(* Logix 5000 project; controller STAT 1756-L72 rev 20.12; software revision 20.04; part 21 of 34 *)
(* tags used below, declared in another part *)
   B10 : DINT[20];
   B14 : DINT[30];
   B17 : DINT[30];
   B3 : DINT[256];
   B9 : DINT[40];
   def1bassin : DINT;
   def2bassin : DINT;
   F8 : REAL[256];
   I10_000_Bit07 : ALIAS FOR I10[0].7;   // Hand Automaat CL8
   I19_000_Bit07 : ALIAS FOR I19[0].7;   // LACK DETECTIE H2SO4
   I1_001_Bit15 : ALIAS FOR I1[1].15;
   I1_008_Bit01 : ALIAS FOR I1[8].1;   // Hand Automaat stormbekken
   I1_016_Bit01 : ALIAS FOR I1[16].1;   // CL2 Hamd /Autom
   I1_017_Bit01 : ALIAS FOR I1[17].1;   // CL3 Hamd /Autom
   I1_018_Bit01 : ALIAS FOR I1[18].1;   // CL4 Hamd /Autom
   I2 : INT[2];
   I3 : INT[2];
   I4 : INT[2];
   I5 : INT[2];
   I6 : INT[2];
   I7 : INT[2];
   I8 : INT[2];
   I9_000_Bit09 : ALIAS FOR I9[0].9;   // Hand_Auto CL7
   N11 : DINT[150];
   N12 : DINT[230];
   N13 : DINT[230];
   N26 : DINT[256];
   N7 : DINT[255];
   O12 : INT[2];
   O13 : INT[2];
   O14 : INT[2];
   O15 : INT[2];
   O18 : INT[2];
   S : INT[164];
   T4 : TIMER[200];
(* ibt, continued *)

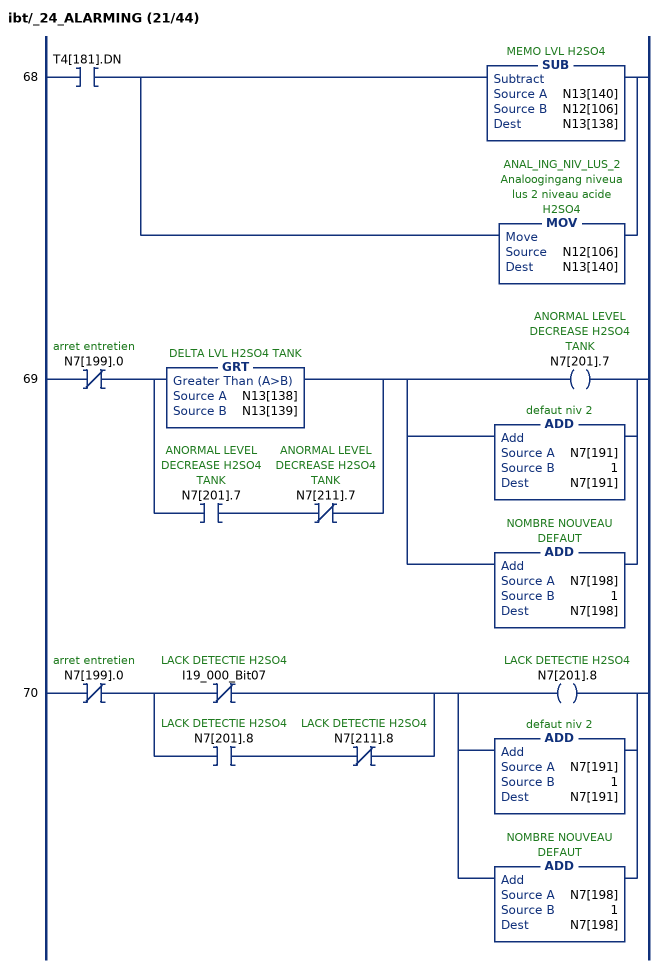
   [picture p391: ibt/_24_ALARMING rungs 68-70]
   68: XIC(T4[181].DN)[SUB(N13[140],N12[106],N13[138]) ,MOV(N12[106],N13[140]) ];
   69: XIO(N7[199].0)[GRT(N13[138],N13[139]) ,XIC(N7[201].7) XIO(N7[211].7) ][OTE(N7[201].7) ,ADD(N7[191],1,N7[191]) ,ADD(N7[198],1,N7[198]) ];
   70: XIO(N7[199].0)[XIO(I19_000_Bit07) ,XIC(N7[201].8) XIO(N7[211].8) ][OTE(N7[201].8) ,ADD(N7[191],1,N7[191]) ,ADD(N7[198],1,N7[198]) ];
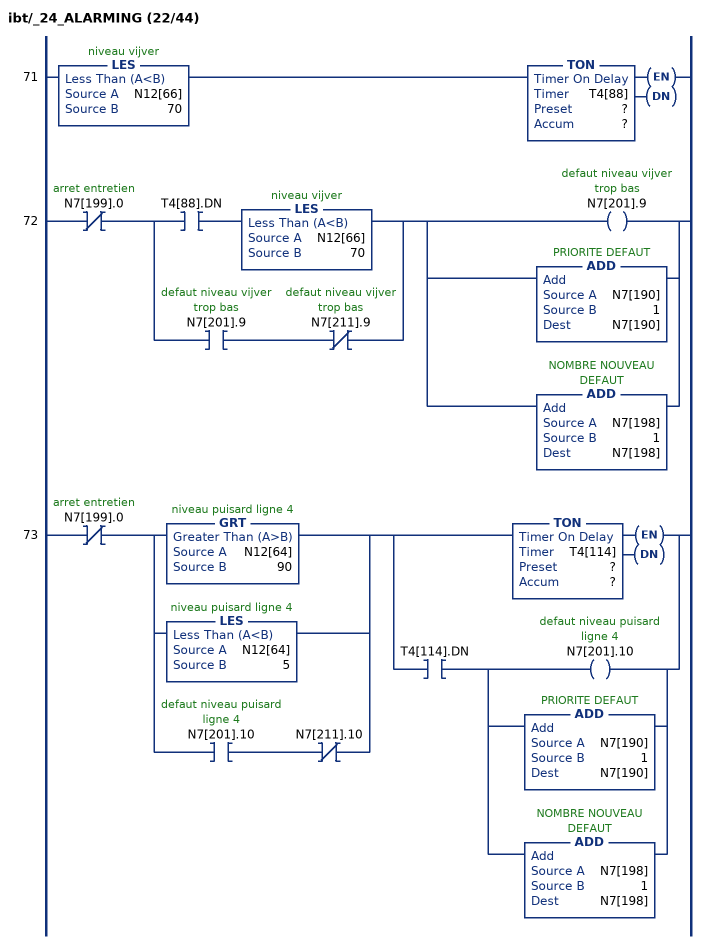
   71: LES(N12[66],70)TON(T4[88],?,?);
   72: XIO(N7[199].0)[XIC(T4[88].DN) LES(N12[66],70) ,XIC(N7[201].9) XIO(N7[211].9) ][OTE(N7[201].9) ,ADD(N7[190],1,N7[190]) ,ADD(N7[198],1,N7[198]) ];
   73: XIO(N7[199].0)[GRT(N12[64],90) ,LES(N12[64],5) ,XIC(N7[201].10) XIO(N7[211].10) ][TON(T4[114],?,?) ,XIC(T4[114].DN) [OTE(N7[201].10) ,ADD(N7[190],1,N7[190]) ,ADD(N7[198],1,N7[198]) ] ];
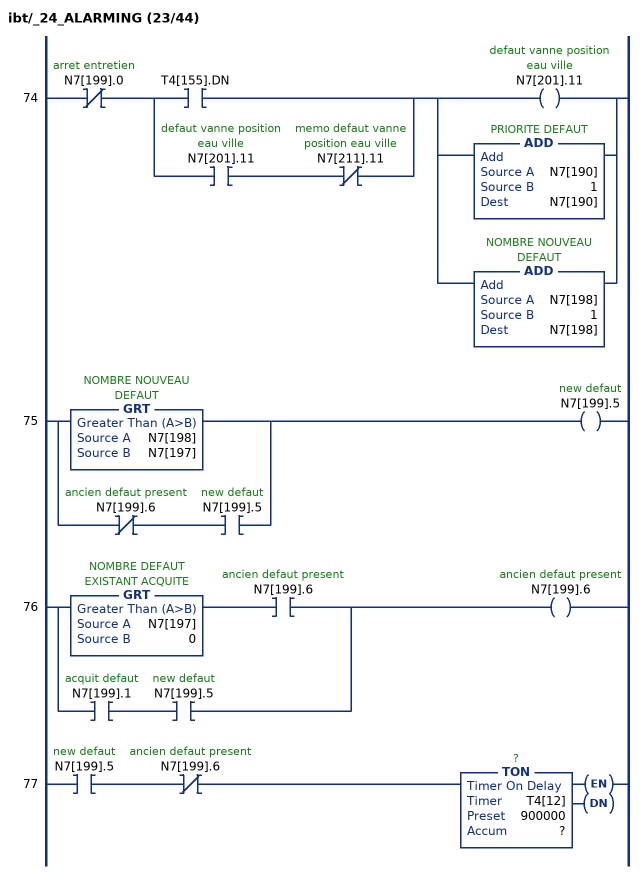
   74: XIO(N7[199].0)[XIC(T4[155].DN) ,XIC(N7[201].11) XIO(N7[211].11) ][OTE(N7[201].11) ,ADD(N7[190],1,N7[190]) ,ADD(N7[198],1,N7[198]) ];
   75: [GRT(N7[198],N7[197]) ,XIO(N7[199].6) XIC(N7[199].5) ]OTE(N7[199].5);
   76: [GRT(N7[197],0) XIC(N7[199].6) ,XIC(N7[199].1) XIC(N7[199].5) ]OTE(N7[199].6);
   77: XIC(N7[199].5)XIO(N7[199].6)TON(T4[12],?,?);
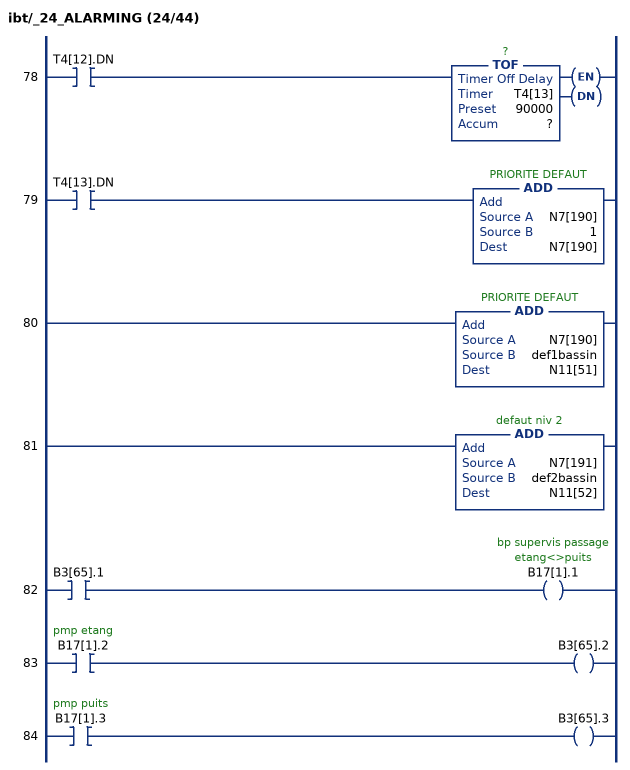
   78: XIC(T4[12].DN)TOF(T4[13],?,?);
   79: XIC(T4[13].DN)ADD(N7[190],1,N7[190]);
   80: ADD(N7[190],def1bassin,N11[51]);
   81: ADD(N7[191],def2bassin,N11[52]);
   82: XIC(B3[65].1)OTE(B17[1].1);
   83: XIC(B17[1].2)OTE(B3[65].2);
   84: XIC(B17[1].3)OTE(B3[65].3);
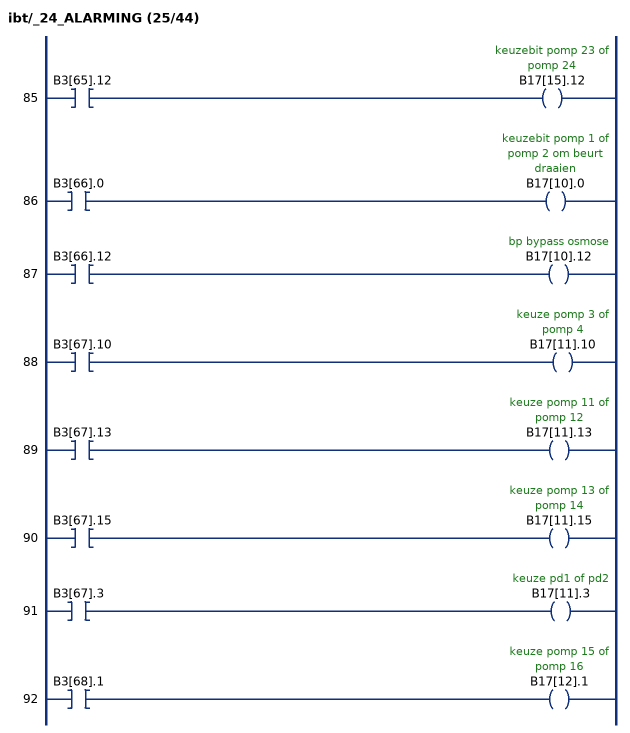
   85: XIC(B3[65].12)OTE(B17[15].12);
   86: XIC(B3[66].0)OTE(B17[10].0);
   87: XIC(B3[66].12)OTE(B17[10].12);
   88: XIC(B3[67].10)OTE(B17[11].10);
   89: XIC(B3[67].13)OTE(B17[11].13);
   90: XIC(B3[67].15)OTE(B17[11].15);
   91: XIC(B3[67].3)OTE(B17[11].3);
   92: XIC(B3[68].1)OTE(B17[12].1);
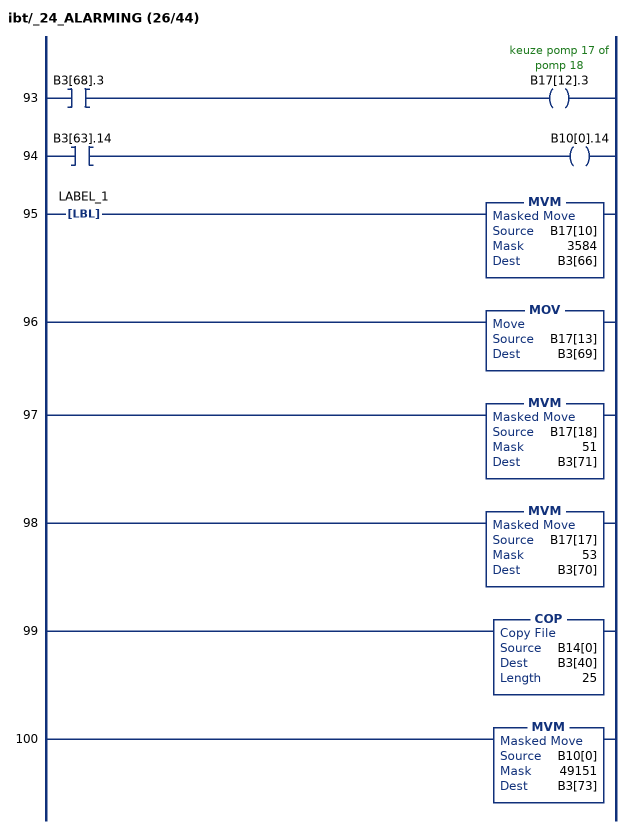
   93: XIC(B3[68].3)OTE(B17[12].3);
   94: XIC(B3[63].14)OTE(B10[0].14);
   95: LBL(LABEL_1)MVM(B17[10],3584,B3[66]);
   96: MOV(B17[13],B3[69]);
   97: MVM(B17[18],51,B3[71]);
   98: MVM(B17[17],53,B3[70]);
   99: COP(B14[0],B3[40],25);
   100: MVM(B10[0],49151,B3[73]);
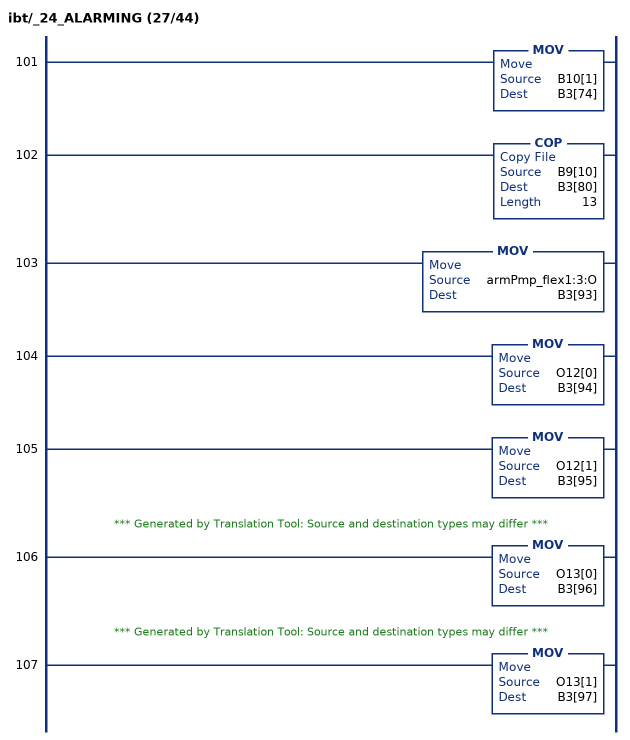
   101: MOV(B10[1],B3[74]);
   102: COP(B9[10],B3[80],13);
   103: MOV(armPmp_flex1:3:O,B3[93]);
   104: MOV(O12[0],B3[94]);
   105: MOV(O12[1],B3[95]);
   // *** Generated by Translation Tool: Source and destination types may differ ***
   106: MOV(O13[0],B3[96]);
   // *** Generated by Translation Tool: Source and destination types may differ ***
   107: MOV(O13[1],B3[97]);
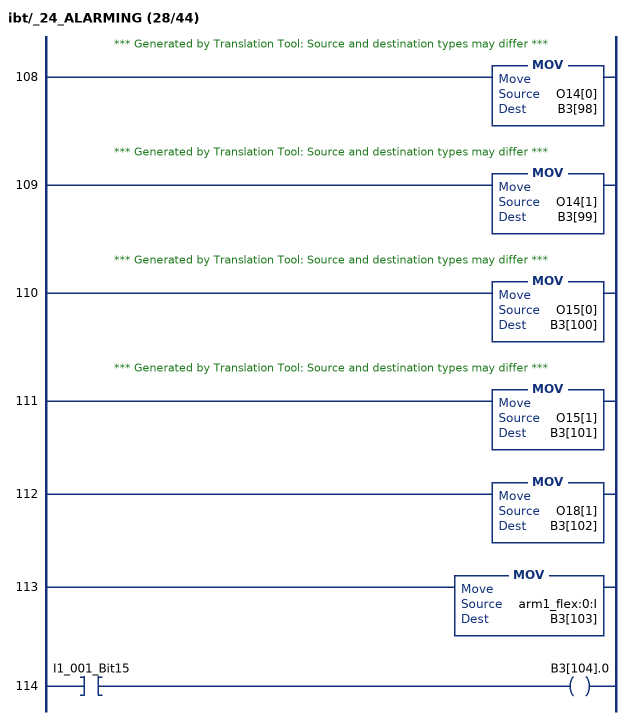
   // *** Generated by Translation Tool: Source and destination types may differ ***
   108: MOV(O14[0],B3[98]);
   // *** Generated by Translation Tool: Source and destination types may differ ***
   109: MOV(O14[1],B3[99]);
   // *** Generated by Translation Tool: Source and destination types may differ ***
   110: MOV(O15[0],B3[100]);
   // *** Generated by Translation Tool: Source and destination types may differ ***
   111: MOV(O15[1],B3[101]);
   112: MOV(O18[1],B3[102]);
   113: MOV(arm1_flex:0:I,B3[103]);
   114: XIC(I1_001_Bit15)OTE(B3[104].0);
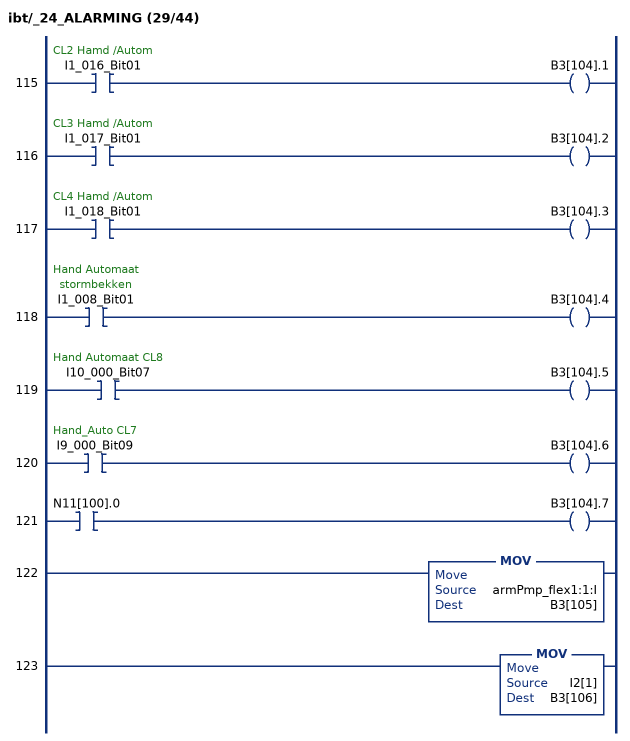
   115: XIC(I1_016_Bit01)OTE(B3[104].1);
   116: XIC(I1_017_Bit01)OTE(B3[104].2);
   117: XIC(I1_018_Bit01)OTE(B3[104].3);
   118: XIC(I1_008_Bit01)OTE(B3[104].4);
   119: XIC(I10_000_Bit07)OTE(B3[104].5);
   120: XIC(I9_000_Bit09)OTE(B3[104].6);
   121: XIC(N11[100].0)OTE(B3[104].7);
   122: MOV(armPmp_flex1:1:I,B3[105]);
   123: MOV(I2[1],B3[106]);
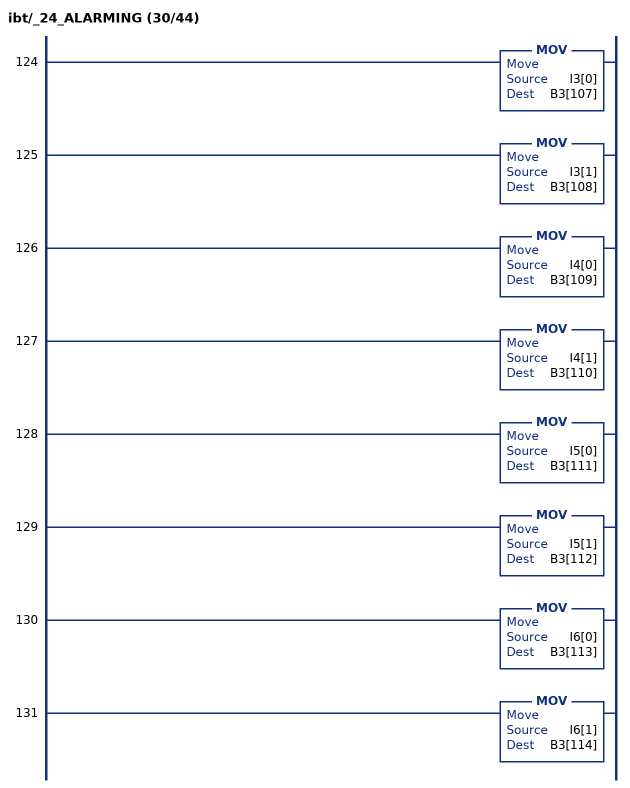
   124: MOV(I3[0],B3[107]);
   125: MOV(I3[1],B3[108]);
   126: MOV(I4[0],B3[109]);
   127: MOV(I4[1],B3[110]);
   128: MOV(I5[0],B3[111]);
   129: MOV(I5[1],B3[112]);
   130: MOV(I6[0],B3[113]);
   131: MOV(I6[1],B3[114]);
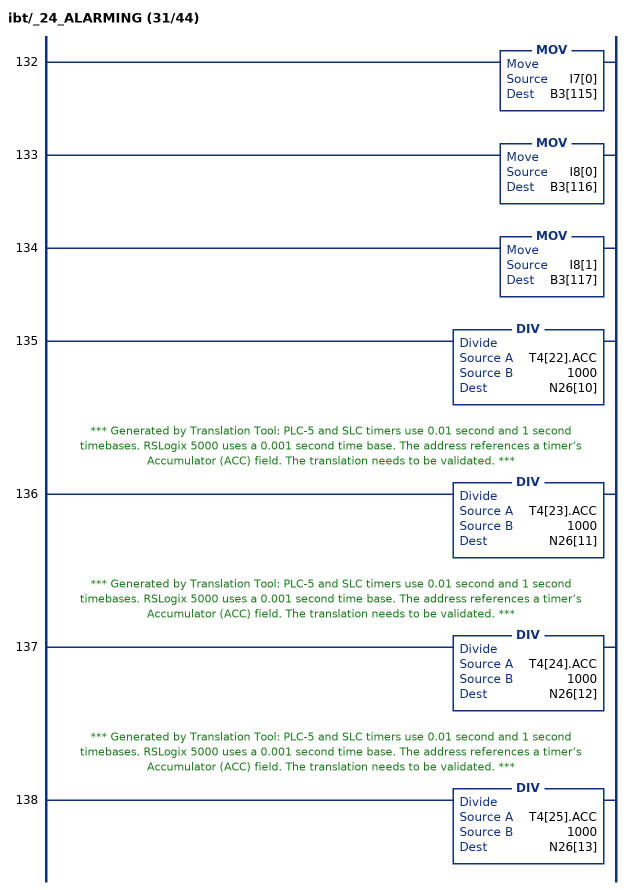
   132: MOV(I7[0],B3[115]);
   133: MOV(I8[0],B3[116]);
   134: MOV(I8[1],B3[117]);
   135: DIV(T4[22].ACC,1000,N26[10]);
   // *** Generated by Translation Tool: PLC-5 and SLC timers use 0.01 second and 1 second timebases. RSLogix 5000 uses a 0.001 second time base. The address references a timer’s Accumulator (ACC) field. The translation needs to be validated. ***
   136: DIV(T4[23].ACC,1000,N26[11]);
   // *** Generated by Translation Tool: PLC-5 and SLC timers use 0.01 second and 1 second timebases. RSLogix 5000 uses a 0.001 second time base. The address references a timer’s Accumulator (ACC) field. The translation needs to be validated. ***
   137: DIV(T4[24].ACC,1000,N26[12]);
   // *** Generated by Translation Tool: PLC-5 and SLC timers use 0.01 second and 1 second timebases. RSLogix 5000 uses a 0.001 second time base. The address references a timer’s Accumulator (ACC) field. The translation needs to be validated. ***
   138: DIV(T4[25].ACC,1000,N26[13]);
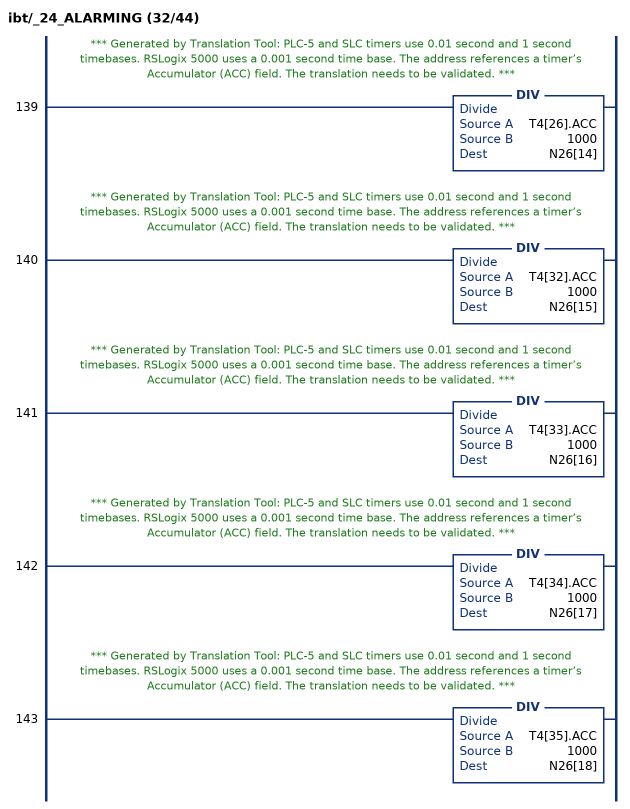
   // *** Generated by Translation Tool: PLC-5 and SLC timers use 0.01 second and 1 second timebases. RSLogix 5000 uses a 0.001 second time base. The address references a timer’s Accumulator (ACC) field. The translation needs to be validated. ***
   139: DIV(T4[26].ACC,1000,N26[14]);
   // *** Generated by Translation Tool: PLC-5 and SLC timers use 0.01 second and 1 second timebases. RSLogix 5000 uses a 0.001 second time base. The address references a timer’s Accumulator (ACC) field. The translation needs to be validated. ***
   140: DIV(T4[32].ACC,1000,N26[15]);
   // *** Generated by Translation Tool: PLC-5 and SLC timers use 0.01 second and 1 second timebases. RSLogix 5000 uses a 0.001 second time base. The address references a timer’s Accumulator (ACC) field. The translation needs to be validated. ***
   141: DIV(T4[33].ACC,1000,N26[16]);
   // *** Generated by Translation Tool: PLC-5 and SLC timers use 0.01 second and 1 second timebases. RSLogix 5000 uses a 0.001 second time base. The address references a timer’s Accumulator (ACC) field. The translation needs to be validated. ***
   142: DIV(T4[34].ACC,1000,N26[17]);
   // *** Generated by Translation Tool: PLC-5 and SLC timers use 0.01 second and 1 second timebases. RSLogix 5000 uses a 0.001 second time base. The address references a timer’s Accumulator (ACC) field. The translation needs to be validated. ***
   143: DIV(T4[35].ACC,1000,N26[18]);
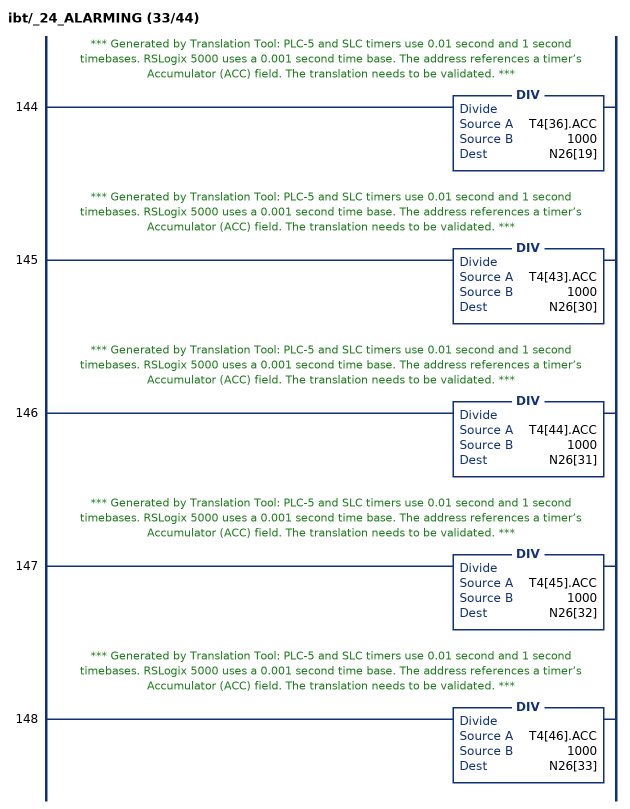
   // *** Generated by Translation Tool: PLC-5 and SLC timers use 0.01 second and 1 second timebases. RSLogix 5000 uses a 0.001 second time base. The address references a timer’s Accumulator (ACC) field. The translation needs to be validated. ***
   144: DIV(T4[36].ACC,1000,N26[19]);
   // *** Generated by Translation Tool: PLC-5 and SLC timers use 0.01 second and 1 second timebases. RSLogix 5000 uses a 0.001 second time base. The address references a timer’s Accumulator (ACC) field. The translation needs to be validated. ***
   145: DIV(T4[43].ACC,1000,N26[30]);
   // *** Generated by Translation Tool: PLC-5 and SLC timers use 0.01 second and 1 second timebases. RSLogix 5000 uses a 0.001 second time base. The address references a timer’s Accumulator (ACC) field. The translation needs to be validated. ***
   146: DIV(T4[44].ACC,1000,N26[31]);
   // *** Generated by Translation Tool: PLC-5 and SLC timers use 0.01 second and 1 second timebases. RSLogix 5000 uses a 0.001 second time base. The address references a timer’s Accumulator (ACC) field. The translation needs to be validated. ***
   147: DIV(T4[45].ACC,1000,N26[32]);
   // *** Generated by Translation Tool: PLC-5 and SLC timers use 0.01 second and 1 second timebases. RSLogix 5000 uses a 0.001 second time base. The address references a timer’s Accumulator (ACC) field. The translation needs to be validated. ***
   148: DIV(T4[46].ACC,1000,N26[33]);
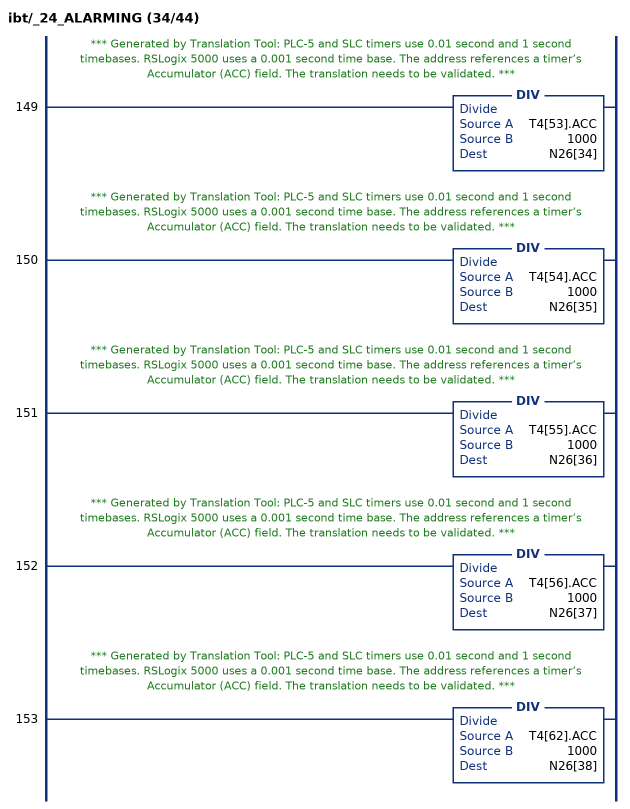
   // *** Generated by Translation Tool: PLC-5 and SLC timers use 0.01 second and 1 second timebases. RSLogix 5000 uses a 0.001 second time base. The address references a timer’s Accumulator (ACC) field. The translation needs to be validated. ***
   149: DIV(T4[53].ACC,1000,N26[34]);
   // *** Generated by Translation Tool: PLC-5 and SLC timers use 0.01 second and 1 second timebases. RSLogix 5000 uses a 0.001 second time base. The address references a timer’s Accumulator (ACC) field. The translation needs to be validated. ***
   150: DIV(T4[54].ACC,1000,N26[35]);
   // *** Generated by Translation Tool: PLC-5 and SLC timers use 0.01 second and 1 second timebases. RSLogix 5000 uses a 0.001 second time base. The address references a timer’s Accumulator (ACC) field. The translation needs to be validated. ***
   151: DIV(T4[55].ACC,1000,N26[36]);
   // *** Generated by Translation Tool: PLC-5 and SLC timers use 0.01 second and 1 second timebases. RSLogix 5000 uses a 0.001 second time base. The address references a timer’s Accumulator (ACC) field. The translation needs to be validated. ***
   152: DIV(T4[56].ACC,1000,N26[37]);
   // *** Generated by Translation Tool: PLC-5 and SLC timers use 0.01 second and 1 second timebases. RSLogix 5000 uses a 0.001 second time base. The address references a timer’s Accumulator (ACC) field. The translation needs to be validated. ***
   153: DIV(T4[62].ACC,1000,N26[38]);
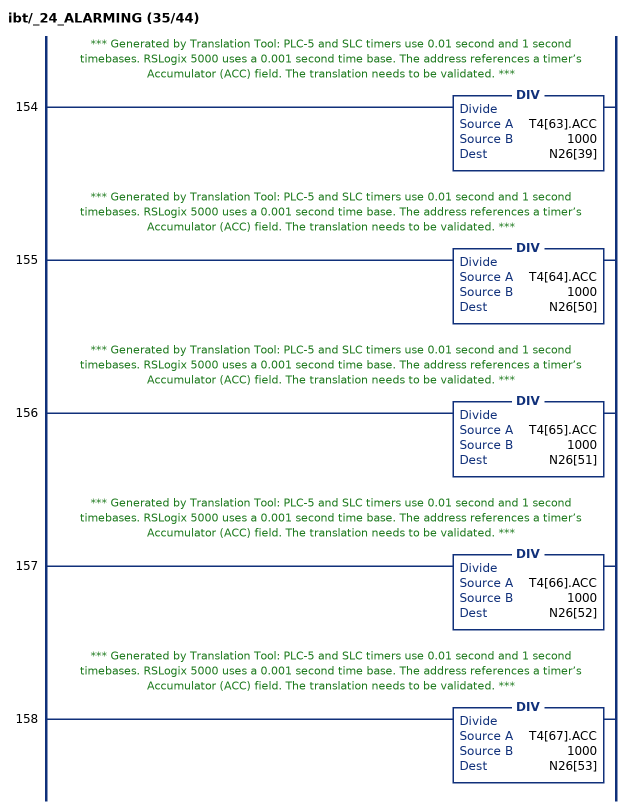
   // *** Generated by Translation Tool: PLC-5 and SLC timers use 0.01 second and 1 second timebases. RSLogix 5000 uses a 0.001 second time base. The address references a timer’s Accumulator (ACC) field. The translation needs to be validated. ***
   154: DIV(T4[63].ACC,1000,N26[39]);
   // *** Generated by Translation Tool: PLC-5 and SLC timers use 0.01 second and 1 second timebases. RSLogix 5000 uses a 0.001 second time base. The address references a timer’s Accumulator (ACC) field. The translation needs to be validated. ***
   155: DIV(T4[64].ACC,1000,N26[50]);
   // *** Generated by Translation Tool: PLC-5 and SLC timers use 0.01 second and 1 second timebases. RSLogix 5000 uses a 0.001 second time base. The address references a timer’s Accumulator (ACC) field. The translation needs to be validated. ***
   156: DIV(T4[65].ACC,1000,N26[51]);
   // *** Generated by Translation Tool: PLC-5 and SLC timers use 0.01 second and 1 second timebases. RSLogix 5000 uses a 0.001 second time base. The address references a timer’s Accumulator (ACC) field. The translation needs to be validated. ***
   157: DIV(T4[66].ACC,1000,N26[52]);
   // *** Generated by Translation Tool: PLC-5 and SLC timers use 0.01 second and 1 second timebases. RSLogix 5000 uses a 0.001 second time base. The address references a timer’s Accumulator (ACC) field. The translation needs to be validated. ***
   158: DIV(T4[67].ACC,1000,N26[53]);
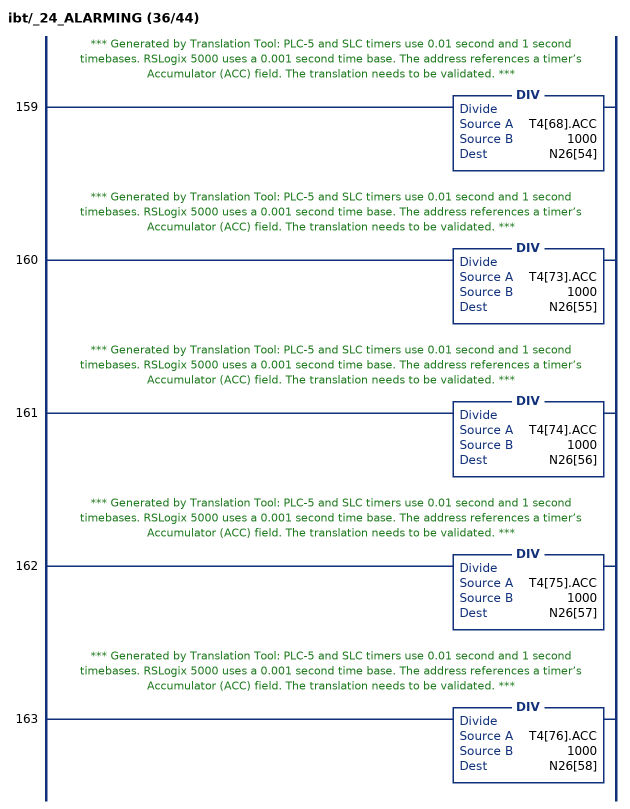
   // *** Generated by Translation Tool: PLC-5 and SLC timers use 0.01 second and 1 second timebases. RSLogix 5000 uses a 0.001 second time base. The address references a timer’s Accumulator (ACC) field. The translation needs to be validated. ***
   159: DIV(T4[68].ACC,1000,N26[54]);
   // *** Generated by Translation Tool: PLC-5 and SLC timers use 0.01 second and 1 second timebases. RSLogix 5000 uses a 0.001 second time base. The address references a timer’s Accumulator (ACC) field. The translation needs to be validated. ***
   160: DIV(T4[73].ACC,1000,N26[55]);
   // *** Generated by Translation Tool: PLC-5 and SLC timers use 0.01 second and 1 second timebases. RSLogix 5000 uses a 0.001 second time base. The address references a timer’s Accumulator (ACC) field. The translation needs to be validated. ***
   161: DIV(T4[74].ACC,1000,N26[56]);
   // *** Generated by Translation Tool: PLC-5 and SLC timers use 0.01 second and 1 second timebases. RSLogix 5000 uses a 0.001 second time base. The address references a timer’s Accumulator (ACC) field. The translation needs to be validated. ***
   162: DIV(T4[75].ACC,1000,N26[57]);
   // *** Generated by Translation Tool: PLC-5 and SLC timers use 0.01 second and 1 second timebases. RSLogix 5000 uses a 0.001 second time base. The address references a timer’s Accumulator (ACC) field. The translation needs to be validated. ***
   163: DIV(T4[76].ACC,1000,N26[58]);
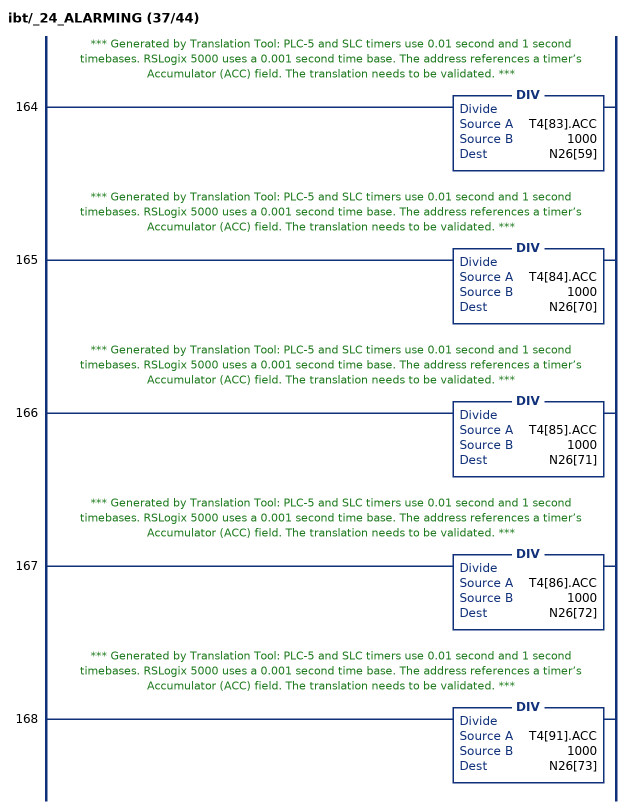
   // *** Generated by Translation Tool: PLC-5 and SLC timers use 0.01 second and 1 second timebases. RSLogix 5000 uses a 0.001 second time base. The address references a timer’s Accumulator (ACC) field. The translation needs to be validated. ***
   164: DIV(T4[83].ACC,1000,N26[59]);
   // *** Generated by Translation Tool: PLC-5 and SLC timers use 0.01 second and 1 second timebases. RSLogix 5000 uses a 0.001 second time base. The address references a timer’s Accumulator (ACC) field. The translation needs to be validated. ***
   165: DIV(T4[84].ACC,1000,N26[70]);
   // *** Generated by Translation Tool: PLC-5 and SLC timers use 0.01 second and 1 second timebases. RSLogix 5000 uses a 0.001 second time base. The address references a timer’s Accumulator (ACC) field. The translation needs to be validated. ***
   166: DIV(T4[85].ACC,1000,N26[71]);
   // *** Generated by Translation Tool: PLC-5 and SLC timers use 0.01 second and 1 second timebases. RSLogix 5000 uses a 0.001 second time base. The address references a timer’s Accumulator (ACC) field. The translation needs to be validated. ***
   167: DIV(T4[86].ACC,1000,N26[72]);
   // *** Generated by Translation Tool: PLC-5 and SLC timers use 0.01 second and 1 second timebases. RSLogix 5000 uses a 0.001 second time base. The address references a timer’s Accumulator (ACC) field. The translation needs to be validated. ***
   168: DIV(T4[91].ACC,1000,N26[73]);
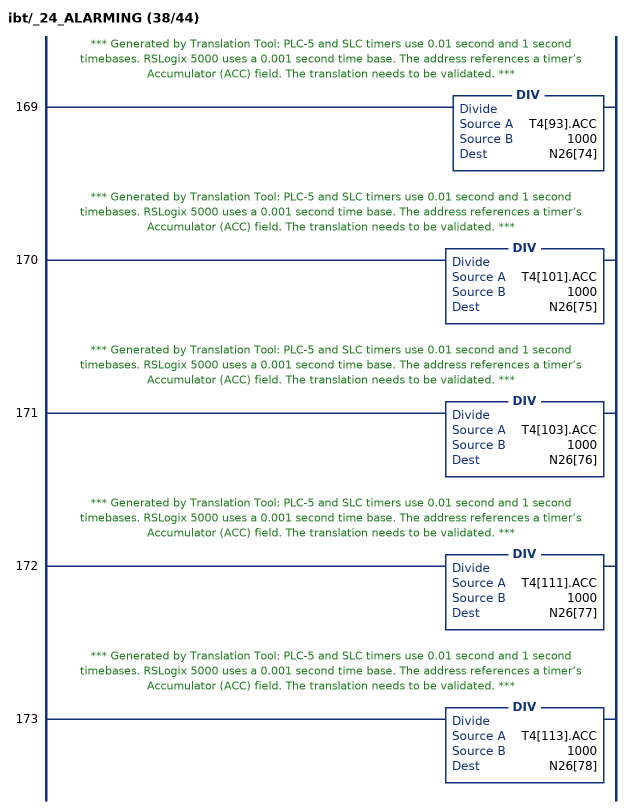
   // *** Generated by Translation Tool: PLC-5 and SLC timers use 0.01 second and 1 second timebases. RSLogix 5000 uses a 0.001 second time base. The address references a timer’s Accumulator (ACC) field. The translation needs to be validated. ***
   169: DIV(T4[93].ACC,1000,N26[74]);
   // *** Generated by Translation Tool: PLC-5 and SLC timers use 0.01 second and 1 second timebases. RSLogix 5000 uses a 0.001 second time base. The address references a timer’s Accumulator (ACC) field. The translation needs to be validated. ***
   170: DIV(T4[101].ACC,1000,N26[75]);
   // *** Generated by Translation Tool: PLC-5 and SLC timers use 0.01 second and 1 second timebases. RSLogix 5000 uses a 0.001 second time base. The address references a timer’s Accumulator (ACC) field. The translation needs to be validated. ***
   171: DIV(T4[103].ACC,1000,N26[76]);
   // *** Generated by Translation Tool: PLC-5 and SLC timers use 0.01 second and 1 second timebases. RSLogix 5000 uses a 0.001 second time base. The address references a timer’s Accumulator (ACC) field. The translation needs to be validated. ***
   172: DIV(T4[111].ACC,1000,N26[77]);
   // *** Generated by Translation Tool: PLC-5 and SLC timers use 0.01 second and 1 second timebases. RSLogix 5000 uses a 0.001 second time base. The address references a timer’s Accumulator (ACC) field. The translation needs to be validated. ***
   173: DIV(T4[113].ACC,1000,N26[78]);
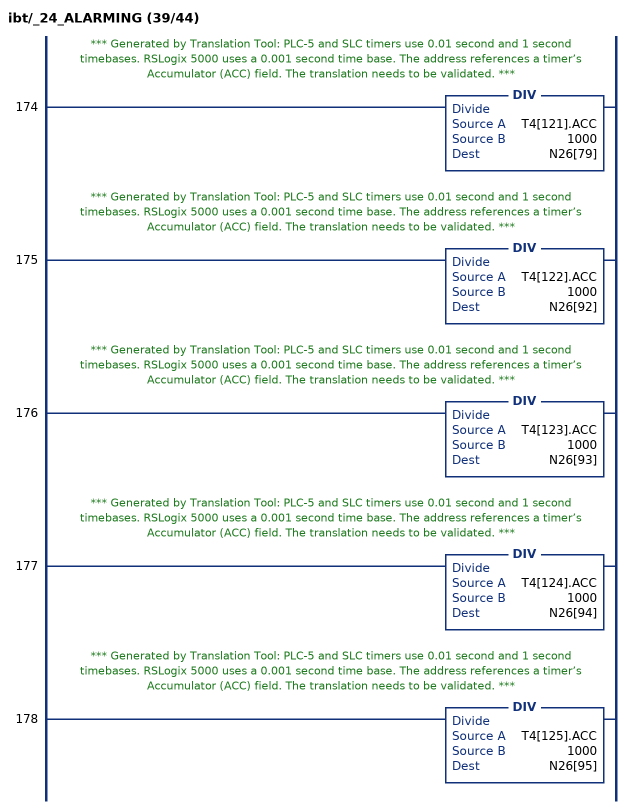
   // *** Generated by Translation Tool: PLC-5 and SLC timers use 0.01 second and 1 second timebases. RSLogix 5000 uses a 0.001 second time base. The address references a timer’s Accumulator (ACC) field. The translation needs to be validated. ***
   174: DIV(T4[121].ACC,1000,N26[79]);
   // *** Generated by Translation Tool: PLC-5 and SLC timers use 0.01 second and 1 second timebases. RSLogix 5000 uses a 0.001 second time base. The address references a timer’s Accumulator (ACC) field. The translation needs to be validated. ***
   175: DIV(T4[122].ACC,1000,N26[92]);
   // *** Generated by Translation Tool: PLC-5 and SLC timers use 0.01 second and 1 second timebases. RSLogix 5000 uses a 0.001 second time base. The address references a timer’s Accumulator (ACC) field. The translation needs to be validated. ***
   176: DIV(T4[123].ACC,1000,N26[93]);
   // *** Generated by Translation Tool: PLC-5 and SLC timers use 0.01 second and 1 second timebases. RSLogix 5000 uses a 0.001 second time base. The address references a timer’s Accumulator (ACC) field. The translation needs to be validated. ***
   177: DIV(T4[124].ACC,1000,N26[94]);
   // *** Generated by Translation Tool: PLC-5 and SLC timers use 0.01 second and 1 second timebases. RSLogix 5000 uses a 0.001 second time base. The address references a timer’s Accumulator (ACC) field. The translation needs to be validated. ***
   178: DIV(T4[125].ACC,1000,N26[95]);
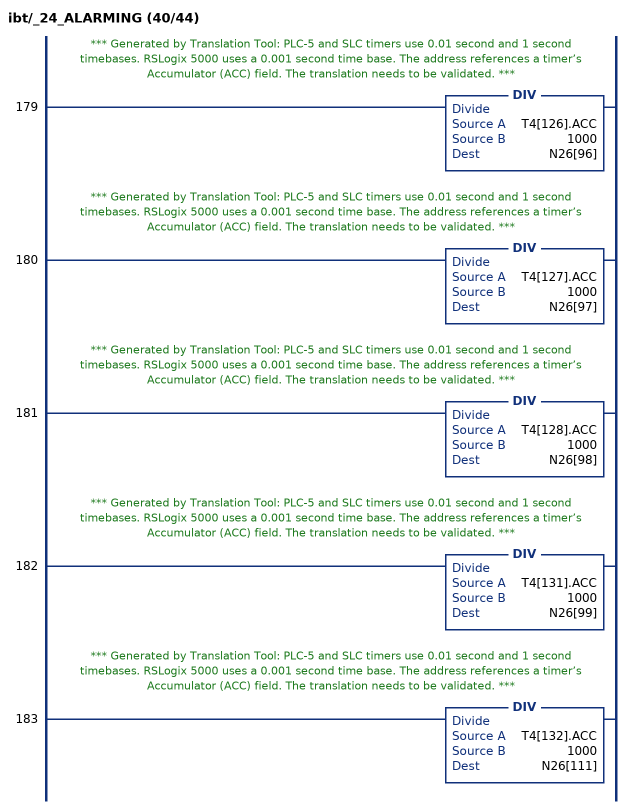
   // *** Generated by Translation Tool: PLC-5 and SLC timers use 0.01 second and 1 second timebases. RSLogix 5000 uses a 0.001 second time base. The address references a timer’s Accumulator (ACC) field. The translation needs to be validated. ***
   179: DIV(T4[126].ACC,1000,N26[96]);
   // *** Generated by Translation Tool: PLC-5 and SLC timers use 0.01 second and 1 second timebases. RSLogix 5000 uses a 0.001 second time base. The address references a timer’s Accumulator (ACC) field. The translation needs to be validated. ***
   180: DIV(T4[127].ACC,1000,N26[97]);
   // *** Generated by Translation Tool: PLC-5 and SLC timers use 0.01 second and 1 second timebases. RSLogix 5000 uses a 0.001 second time base. The address references a timer’s Accumulator (ACC) field. The translation needs to be validated. ***
   181: DIV(T4[128].ACC,1000,N26[98]);
   // *** Generated by Translation Tool: PLC-5 and SLC timers use 0.01 second and 1 second timebases. RSLogix 5000 uses a 0.001 second time base. The address references a timer’s Accumulator (ACC) field. The translation needs to be validated. ***
   182: DIV(T4[131].ACC,1000,N26[99]);
   // *** Generated by Translation Tool: PLC-5 and SLC timers use 0.01 second and 1 second timebases. RSLogix 5000 uses a 0.001 second time base. The address references a timer’s Accumulator (ACC) field. The translation needs to be validated. ***
   183: DIV(T4[132].ACC,1000,N26[111]);
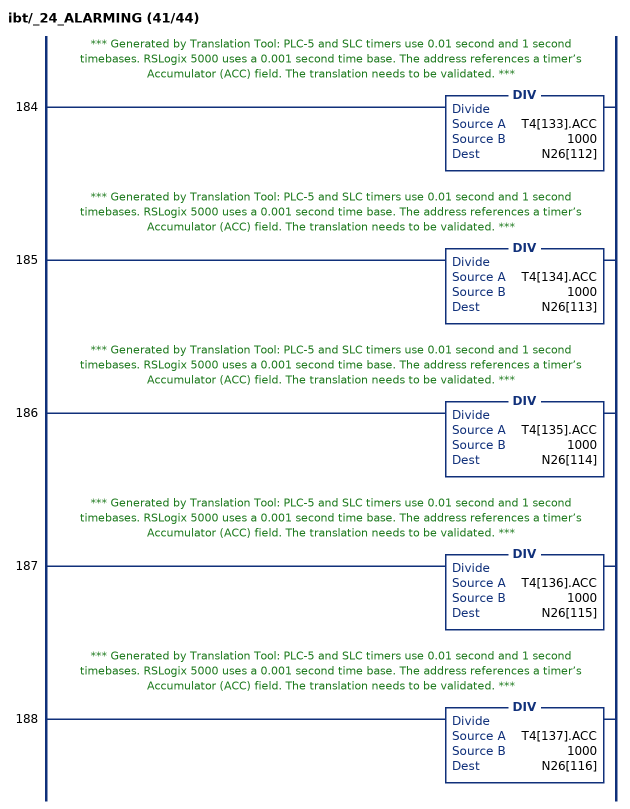
   // *** Generated by Translation Tool: PLC-5 and SLC timers use 0.01 second and 1 second timebases. RSLogix 5000 uses a 0.001 second time base. The address references a timer’s Accumulator (ACC) field. The translation needs to be validated. ***
   184: DIV(T4[133].ACC,1000,N26[112]);
   // *** Generated by Translation Tool: PLC-5 and SLC timers use 0.01 second and 1 second timebases. RSLogix 5000 uses a 0.001 second time base. The address references a timer’s Accumulator (ACC) field. The translation needs to be validated. ***
   185: DIV(T4[134].ACC,1000,N26[113]);
   // *** Generated by Translation Tool: PLC-5 and SLC timers use 0.01 second and 1 second timebases. RSLogix 5000 uses a 0.001 second time base. The address references a timer’s Accumulator (ACC) field. The translation needs to be validated. ***
   186: DIV(T4[135].ACC,1000,N26[114]);
   // *** Generated by Translation Tool: PLC-5 and SLC timers use 0.01 second and 1 second timebases. RSLogix 5000 uses a 0.001 second time base. The address references a timer’s Accumulator (ACC) field. The translation needs to be validated. ***
   187: DIV(T4[136].ACC,1000,N26[115]);
   // *** Generated by Translation Tool: PLC-5 and SLC timers use 0.01 second and 1 second timebases. RSLogix 5000 uses a 0.001 second time base. The address references a timer’s Accumulator (ACC) field. The translation needs to be validated. ***
   188: DIV(T4[137].ACC,1000,N26[116]);
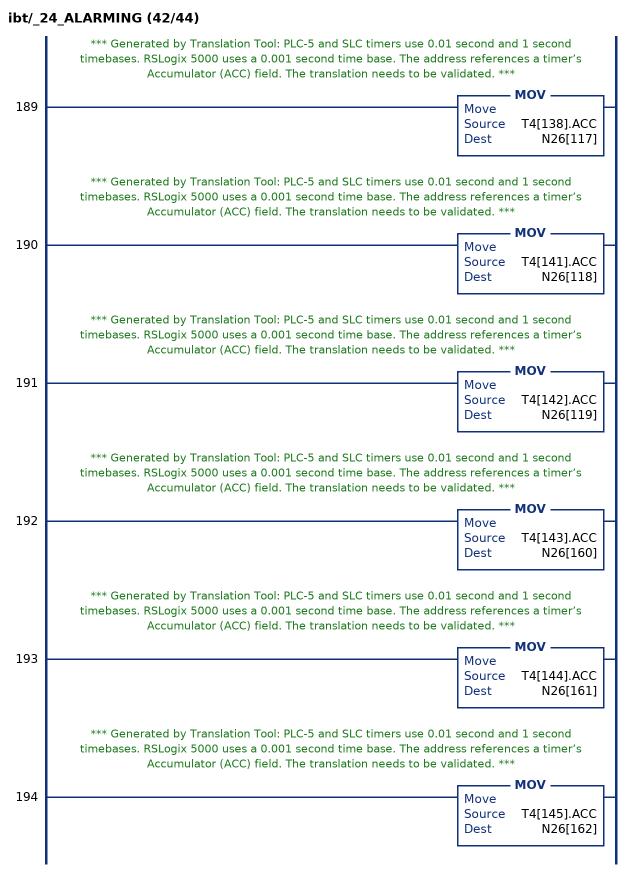
   // *** Generated by Translation Tool: PLC-5 and SLC timers use 0.01 second and 1 second timebases. RSLogix 5000 uses a 0.001 second time base. The address references a timer’s Accumulator (ACC) field. The translation needs to be validated. ***
   189: MOV(T4[138].ACC,N26[117]);
   // *** Generated by Translation Tool: PLC-5 and SLC timers use 0.01 second and 1 second timebases. RSLogix 5000 uses a 0.001 second time base. The address references a timer’s Accumulator (ACC) field. The translation needs to be validated. ***
   190: MOV(T4[141].ACC,N26[118]);
   // *** Generated by Translation Tool: PLC-5 and SLC timers use 0.01 second and 1 second timebases. RSLogix 5000 uses a 0.001 second time base. The address references a timer’s Accumulator (ACC) field. The translation needs to be validated. ***
   191: MOV(T4[142].ACC,N26[119]);
   // *** Generated by Translation Tool: PLC-5 and SLC timers use 0.01 second and 1 second timebases. RSLogix 5000 uses a 0.001 second time base. The address references a timer’s Accumulator (ACC) field. The translation needs to be validated. ***
   192: MOV(T4[143].ACC,N26[160]);
   // *** Generated by Translation Tool: PLC-5 and SLC timers use 0.01 second and 1 second timebases. RSLogix 5000 uses a 0.001 second time base. The address references a timer’s Accumulator (ACC) field. The translation needs to be validated. ***
   193: MOV(T4[144].ACC,N26[161]);
   // *** Generated by Translation Tool: PLC-5 and SLC timers use 0.01 second and 1 second timebases. RSLogix 5000 uses a 0.001 second time base. The address references a timer’s Accumulator (ACC) field. The translation needs to be validated. ***
   194: MOV(T4[145].ACC,N26[162]);
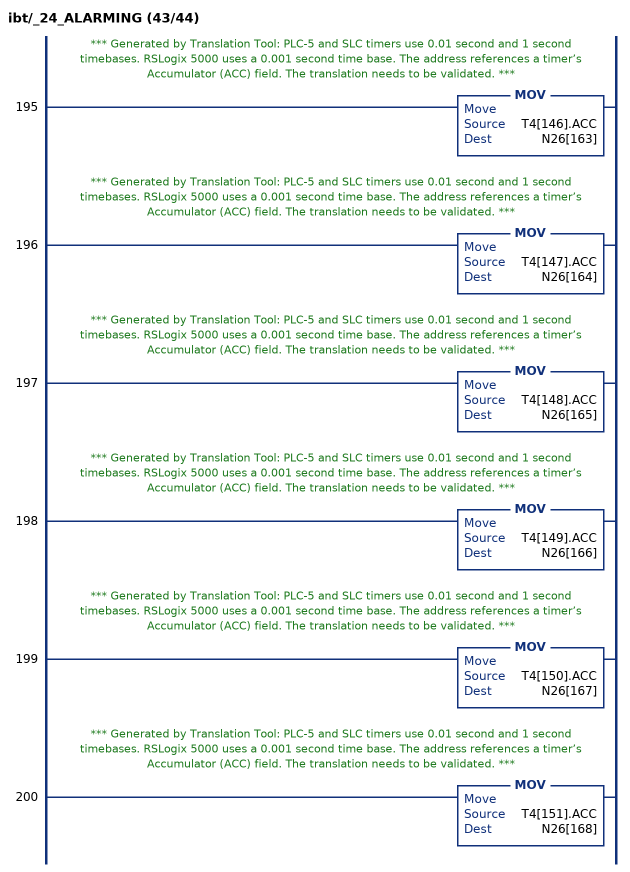
   // *** Generated by Translation Tool: PLC-5 and SLC timers use 0.01 second and 1 second timebases. RSLogix 5000 uses a 0.001 second time base. The address references a timer’s Accumulator (ACC) field. The translation needs to be validated. ***
   195: MOV(T4[146].ACC,N26[163]);
   // *** Generated by Translation Tool: PLC-5 and SLC timers use 0.01 second and 1 second timebases. RSLogix 5000 uses a 0.001 second time base. The address references a timer’s Accumulator (ACC) field. The translation needs to be validated. ***
   196: MOV(T4[147].ACC,N26[164]);
   // *** Generated by Translation Tool: PLC-5 and SLC timers use 0.01 second and 1 second timebases. RSLogix 5000 uses a 0.001 second time base. The address references a timer’s Accumulator (ACC) field. The translation needs to be validated. ***
   197: MOV(T4[148].ACC,N26[165]);
   // *** Generated by Translation Tool: PLC-5 and SLC timers use 0.01 second and 1 second timebases. RSLogix 5000 uses a 0.001 second time base. The address references a timer’s Accumulator (ACC) field. The translation needs to be validated. ***
   198: MOV(T4[149].ACC,N26[166]);
   // *** Generated by Translation Tool: PLC-5 and SLC timers use 0.01 second and 1 second timebases. RSLogix 5000 uses a 0.001 second time base. The address references a timer’s Accumulator (ACC) field. The translation needs to be validated. ***
   199: MOV(T4[150].ACC,N26[167]);
   // *** Generated by Translation Tool: PLC-5 and SLC timers use 0.01 second and 1 second timebases. RSLogix 5000 uses a 0.001 second time base. The address references a timer’s Accumulator (ACC) field. The translation needs to be validated. ***
   200: MOV(T4[151].ACC,N26[168]);
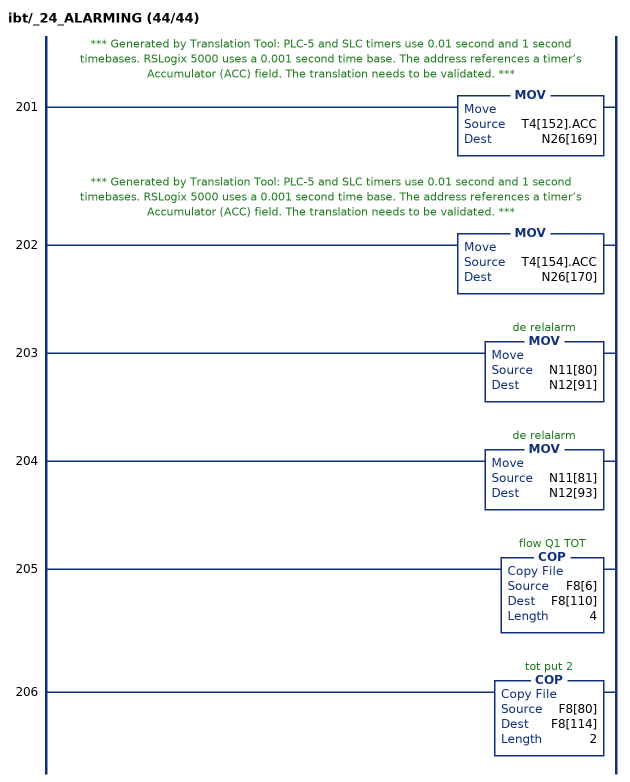
   // *** Generated by Translation Tool: PLC-5 and SLC timers use 0.01 second and 1 second timebases. RSLogix 5000 uses a 0.001 second time base. The address references a timer’s Accumulator (ACC) field. The translation needs to be validated. ***
   201: MOV(T4[152].ACC,N26[169]);
   // *** Generated by Translation Tool: PLC-5 and SLC timers use 0.01 second and 1 second timebases. RSLogix 5000 uses a 0.001 second time base. The address references a timer’s Accumulator (ACC) field. The translation needs to be validated. ***
   202: MOV(T4[154].ACC,N26[170]);
   203: MOV(N11[80],N12[91]);
   204: MOV(N11[81],N12[93]);
   205: COP(F8[6],F8[110],4);
   206: COP(F8[80],F8[114],2);
END_ROUTINE
